// TIA Portal V20 export
TYPE "TypeLinmotRd"
   STRUCT
      StatVar : Struct   // State Var
         SubState : Byte;   // main state
         MainState : Byte;   // sub state
      END_STRUCT;
      StatWord : Struct   // Status Word
         OperationEnabled : Bool;   // 1 = State Nr 8 or higher (copied to drive EN LED )
         SwitchOnActive : Bool;   // 1 = Control Word Bit 0
         EnableOperation : Bool;   // 1 = Control Word Bit 3
         Error : Bool;   // 1 = Error
         VoltageEnable : Bool;   // 1 = Control Word Bit 1
         QuickStop : Bool;   // 1 = Control Word Bit 2
         SwitchOnLocked : Bool;   // 1= Release with 0 of Control word bit 0 (Switch On)
         Warning : Bool;   // 1 = One or more bits in the Warn Word are set
         EventHandlerActive : Bool;   // Event Handler setup
         SpecialMotionActive : Bool;   // Special motion commands (Homing, ..) runs
         InTargetPosition : Bool;   // Actual position after motion in window
         Homed : Bool;   // Position sensor system valid
         FatalError : Bool;   // A fatal error can not be acknowledged!
         MotionActive : Bool;   // Setpoint generation (VAI, curve) active
         RangeIndicator1 : Bool;   // Defined UPID is in Range 1
         RangeIndicator2 : Bool;   // Defined UPID is in Range 2
      END_STRUCT;
      WarnWord : Struct   // Warning Word
         MotorHotSensor : Bool;
         MotorShortTimerOverload : Bool;
         MotorSupplyVoltageLow : Bool;
         MotorSupplyVoltageHigh : Bool;
         PositionLagAlways : Bool;
         Res5 : Bool;
         DriveHot : Bool;
         MotorNotHomed : Bool;
         PTC_Sensor1Hot : Bool;
         PTC_Sensor2Hot : Bool;
         Res10 : Bool;
         Res11 : Bool;
         Res12 : Bool;
         Res13 : Bool;
         InterfaceWarnFlag : Bool;
         ApplicationWarnFlag : Bool;
      END_STRUCT;
      Tarpos : DInt;   // target position
      Actpos : DInt;   // actual position
      TarCurrent : DInt;   // target current
      CfgStatWord : Int;   // config status word
      CfgId : Int;   // config index response
      CfgVal : DInt;   // config value response
   END_STRUCT;
END_TYPE
